// Allocates memory for T_Generic.
FUNCTION F_Malloc_Generic : POINTER TO T_Generic
VAR_INPUT
	Count : T_Capacity;
END_VAR
VAR_OUTPUT
	bSuccess : BOOL;
	Error : T_Error := GVL_Errors.ERR_NO_ERROR;
END_VAR
VAR
	Size : UDINT;
END_VAR

Size := TO_UDINT(SIZEOF(T_Generic) * Count);
F_Malloc_Generic := __NEW(BYTE, Size);

IF F_Malloc_Generic = 0 THEN 
	Error := GVL_Errors.ERR_MALLOC_FAILED;
	RETURN;
	END_IF
	
F_Malloc_Generic^.TypeClass := T_Type.TYPE_NONE;
bSuccess := TRUE;

END_FUNCTION

(* stored: Version 1.1.0.1
   POU F_Malloc_Generic: Id {6c6e9db2-79b4-08ab-287d-97b12703691a}, SpecialFunc None *)
